FUNCTION_BLOCK TURNTABLE_MODEL (* Basic Function Block Type *)
  (* Standard: 61499-2 *)
  (* Version 0.3, 2009-09-15, JHC, Holobloc Inc, Changed transition priorities. *)
  (* Version 0.2, 2003-12-04, JHC, Rockwell Automation, Renamed for better indexing. *)
  (* Version 0.1, 2002-11-05, JHC, Rockwell Automation, Corrected missing ST element in Algorithm REQ. *)
  (* Version 0.0, 2000-05-30, JHC, Rockwell Automation *)
  PACKAGE fb.rt.Conveyer;
  IMPORT fb.datatype.*;
  IMPORT fb.rt.*;
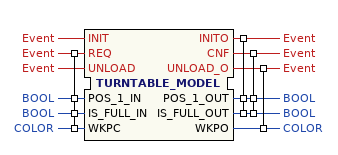
  EVENT_INPUT
    INIT; (* Initialization Request *)
    REQ WITH POS_1_IN, IS_FULL_IN, WKPC; (* Normal Execution Request *)
    UNLOAD;
  END_EVENT
  EVENT_OUTPUT
    INITO WITH POS_1_OUT, IS_FULL_OUT; (* Initialization Confirm *)
    CNF WITH POS_1_OUT, IS_FULL_OUT; (* Execution Confirmation *)
    UNLOAD_O WITH WKPO;
  END_EVENT
  VAR_INPUT
    POS_1_IN : BOOL;
    IS_FULL_IN : BOOL;
    WKPC : COLOR;
  END_VAR
  VAR_OUTPUT
    POS_1_OUT : BOOL;
    IS_FULL_OUT : BOOL;
    WKPO : COLOR;
  END_VAR
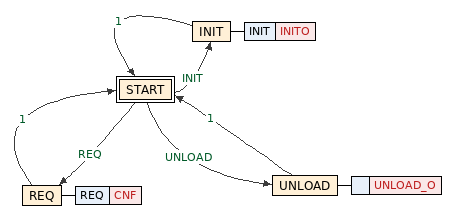
  EC_STATES
    START; (* Initial State *)
    INIT : INIT -> INITO; (* Initialization *)
    REQ : REQ -> CNF; (* Normal execution *)
    UNLOAD : -> UNLOAD_O;
  END_STATES
  EC_TRANSITIONS
    INIT TO START := 1;
    START TO REQ := REQ;
    START TO INIT := INIT;
    REQ TO START := 1;
    START TO UNLOAD := UNLOAD;
    UNLOAD TO START := 1;
  END_TRANSITIONS
  ALGORITHM INIT IN ST: (* Initialization algorithm *)
POS_1_IN := TRUE;
IS_FULL_IN := FALSE;
POS_1_OUT := TRUE;
IS_FULL_OUT := FALSE;
  END_ALGORITHM
  ALGORITHM REQ IN ST: (* Normally executed algorithm *)
POS_1_OUT := POS_1_IN;
IS_FULL_OUT := IS_FULL_IN;
WKPO := WKPC;
  END_ALGORITHM
END_FUNCTION_BLOCK
